% RSLogix 500 project P1_BAK000.RSS, saved by version 8.30.00.16 %
PROJECT "UNTITLED"    % processor: Bul.1763 MicroLogix 1100 Series B %

PROGRAM FILES
  LAD 2 "MAIN"  3 rungs
  LAD 3 "DIGITALI/O"  5 rungs
  LAD 4 "CONTROLS"  11 rungs

DATA FILES
  O0 OUTPUT  4 elements
  I1 INPUT  6 elements
  S2 STATUS  66 elements
  B3 BINARY  1 elements
  T4 TIMER  1 elements
  C5 COUNTER  1 elements
  R6 CONTROL  1 elements
  N7 INTEGER  1 elements
  F8 FLOAT  1 elements

LADDER 2 "MAIN"
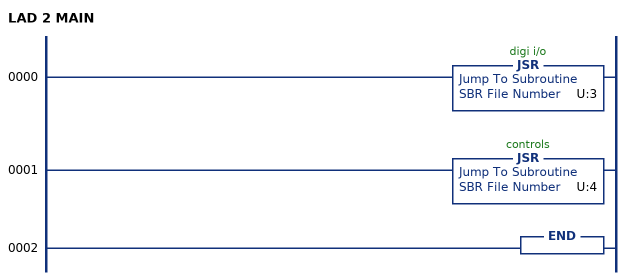
% Rung: 0 %  % edit flag set %
SOR JSR U:3 EOR
%   U:3  "digi i/o" %
% Rung: 1 %  % edit flag set %
SOR JSR U:4 EOR
%   U:4  "controls" %
% Rung: 2 %
SOR END EOR

LADDER 3 "DIGITALI/O"
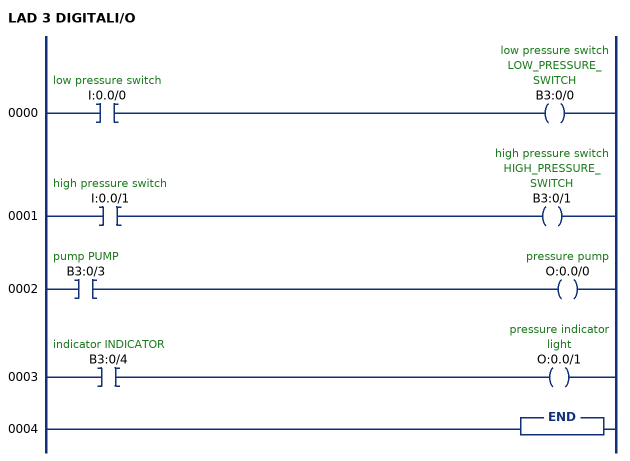
% Rung: 0 %  % edit flag set %
SOR XIC I:0.0/0 OTE B3:0/0 EOR
%   I:0.0/0  "low pressure switch" %
%   B3:0/0  LOW_PRESSURE_SWITCH  "low pressure switch" %
% Rung: 1 %  % edit flag set %
SOR XIC I:0.0/1 OTE B3:0/1 EOR
%   I:0.0/1  "high pressure switch" %
%   B3:0/1  HIGH_PRESSURE_SWITCH  "high pressure switch" %
% Rung: 2 %  % edit flag set %
SOR XIC B3:0/3 OTE O:0.0/0 EOR
%   B3:0/3  PUMP  "pump" %
%   O:0.0/0  "pressure pump" %
% Rung: 3 %  % edit flag set %
SOR XIC B3:0/4 OTE O:0.0/1 EOR
%   B3:0/4  INDICATOR  "indicator" %
%   O:0.0/1  "pressure indicator light" %
% Rung: 4 %
SOR END EOR

LADDER 4 "CONTROLS"
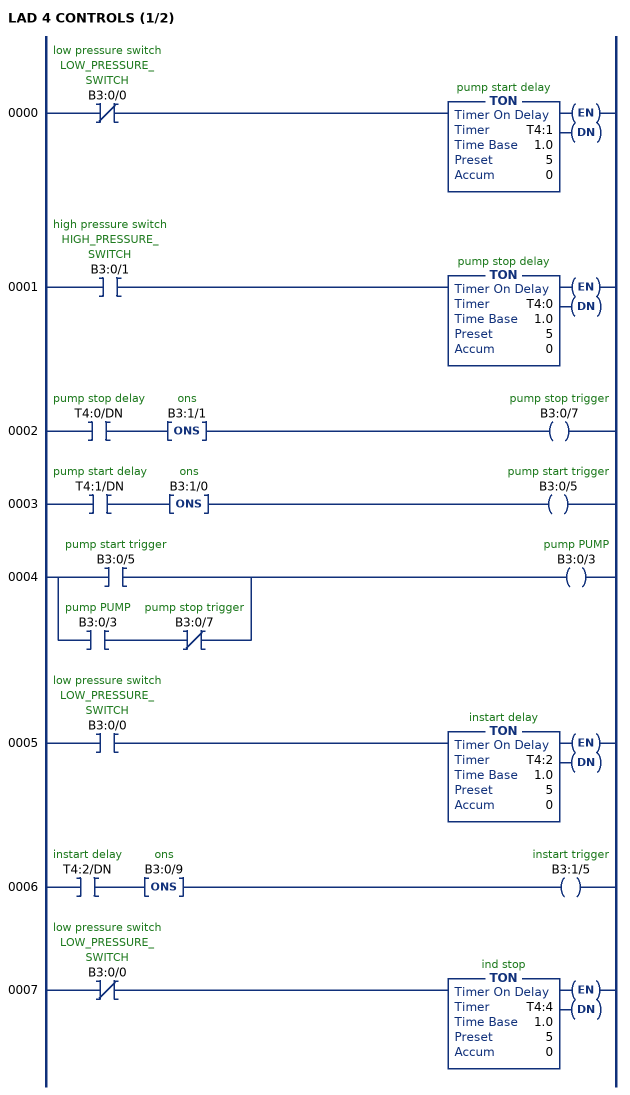
% Rung: 0 %  % edit flag set %
SOR XIO B3:0/0 TON T4:1 1.0 5 0 EOR
%   B3:0/0  LOW_PRESSURE_SWITCH  "low pressure switch" %
%   T4:1  "pump start delay" %
% Rung: 1 %  % edit flag set %
SOR XIC B3:0/1 TON T4:0 1.0 5 0 EOR
%   B3:0/1  HIGH_PRESSURE_SWITCH  "high pressure switch" %
%   T4:0  "pump stop delay" %
% Rung: 2 %  % edit flag set %
SOR XIC T4:0/DN ONS B3:1/1 OTE B3:0/7 EOR
%   T4:0/DN  "pump stop delay" %
%   B3:1/1  "ons" %
%   B3:0/7  "pump stop trigger" %
% Rung: 3 %  % edit flag set %
SOR XIC T4:1/DN ONS B3:1/0 OTE B3:0/5 EOR
%   T4:1/DN  "pump start delay" %
%   B3:1/0  "ons" %
%   B3:0/5  "pump start trigger" %
% Rung: 4 %  % edit flag set %
SOR BST XIC B3:0/5 NXB XIC B3:0/3 XIO B3:0/7 BND OTE B3:0/3 EOR
%   B3:0/5  "pump start trigger" %
%   B3:0/3  PUMP  "pump" %
%   B3:0/7  "pump stop trigger" %
% Rung: 5 %  % edit flag set %
SOR XIC B3:0/0 TON T4:2 1.0 5 0 EOR
%   B3:0/0  LOW_PRESSURE_SWITCH  "low pressure switch" %
%   T4:2  "instart delay" %
% Rung: 6 %  % edit flag set %
SOR XIC T4:2/DN ONS B3:0/9 OTE B3:1/5 EOR
%   T4:2/DN  "instart delay" %
%   B3:0/9  "ons" %
%   B3:1/5  "instart trigger" %
% Rung: 7 %  % edit flag set %
SOR XIO B3:0/0 TON T4:4 1.0 5 0 EOR
%   B3:0/0  LOW_PRESSURE_SWITCH  "low pressure switch" %
%   T4:4  "ind stop" %

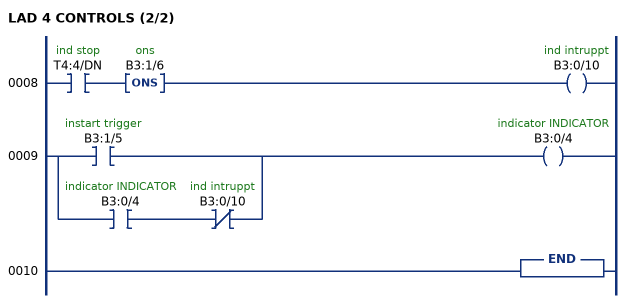
% Rung: 8 %  % edit flag set %
SOR XIC T4:4/DN ONS B3:1/6 OTE B3:0/10 EOR
%   T4:4/DN  "ind stop" %
%   B3:1/6  "ons" %
%   B3:0/10  "ind intruppt" %
% Rung: 9 %  % edit flag set %
SOR BST XIC B3:1/5 NXB XIC B3:0/4 XIO B3:0/10 BND OTE B3:0/4 EOR
%   B3:1/5  "instart trigger" %
%   B3:0/4  INDICATOR  "indicator" %
%   B3:0/10  "ind intruppt" %
% Rung: 10 %
SOR END EOR
